(* PLC project 03_ParoEmergencia.project, CODESYS CODESYS V3.5 SP22 Patch 3 *)
(* stored: creationDateTime 2026-08-12T12:56:38.0927994, modificationDateTime 2026-08-11T17:50:14.3207698 *)

PROGRAM PLC_PRG
  VAR
    xMarcha : BOOL;
    xMotor : BOOL;
    xParo : BOOL;
    xSeta : BOOL;
  END_VAR

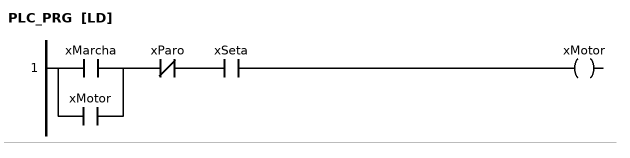
(* LD diagram, written out as Structured Text *)

xMotor := (xMarcha OR xMotor) AND NOT xParo AND xSeta;
END_PROGRAM

CONFIGURATION Device
  RESOURCE Application ON PLC
    TASK MainTask(INTERVAL := T#20ms, PRIORITY := 1);
    PROGRAM PLC_PRG WITH MainTask : PLC_PRG;
  END_RESOURCE
END_CONFIGURATION
